FUNCTION_BLOCK FB_EpicsMeasurement
VAR_INPUT
	InterlockActive_IN : BOOL;
END_VAR
VAR_OUTPUT
	Interlock : BOOL;
	MeasurementValue_OUT : LREAL;
END_VAR
VAR
	MeasurementValue : LREAL;
	MeasurementLowThreshold : LREAL;
	MeasurementHighThreshold : LREAL;
	State : E_EpicsMeasurementState;
	ConnectionTimer : TON;
	Timeout : TIME := T#1.2S;
END_VAR

IF State <> E_EpicsMeasurementState.isOkay AND State <> E_EpicsMeasurementState.isInactive THEN
	Interlock := FALSE;
END_IF

IF InterlockActive_IN THEN
	IF  MeasurementValue > CONSTANTS.MINIMUM_LREAL_THRESHOLD THEN
		MeasurementValue_OUT := MeasurementValue;
		IF MeasurementValue < MeasurementLowThreshold OR MeasurementValue > MeasurementHighThreshold THEN
			State := E_EpicsMeasurementState.isOutOfRange;
		END_IF
		MeasurementValue := CONSTANTS.MINIMUM_LREAL;
		ConnectionTimer(IN := FALSE);
	ELSE
		ConnectionTimer(IN := TRUE);
	END_IF
	
	ConnectionTimer(PT := Timeout);
	
	IF ConnectionTimer.Q THEN
		State := E_EpicsMeasurementState.hasTimeout;	
	END_IF
ELSE
	State := E_EpicsMeasurementState.isInactive;
END_IF

METHOD Acknowledge : BOOL
VAR_INPUT
END_VAR
Interlock := TRUE;
State := E_EpicsMeasurementState.isOkay;
ConnectionTimer(IN := FALSE);
END_METHOD

METHOD Control : BOOL
VAR_IN_OUT
	structure : ST_EpicsMeasurement;
END_VAR
MeasurementValue := structure.MeasurementValueSt;
structure.InterlockSt := Interlock;
MeasurementLowThreshold := structure.MeasurementLowThresholdSt;
MeasurementHighThreshold := structure.MeasurementHighThresholdSt;
structure.MeasurementValueSt := CONSTANTS.MINIMUM_LREAL;
END_METHOD

END_FUNCTION_BLOCK

(* stored: Version 1.1.0.1, ProductVersion 3.1.4024.12
   POU FB_EpicsMeasurement: Id {c62d77d7-8e70-4bc1-ba22-64985e093039}, SpecialFunc None
   Method Acknowledge: Id {2f37e7c4-adc7-4eed-8844-ee69afdbf18f}
   Method Control: Id {56378782-c85a-483a-80f3-9a480c56e45f} *)
